PROGRAM MAIN
VAR
	bStartStop: BOOL := FALSE;
  bReset:     BOOL := FALSE;
  iCounter:   UINT := 0;
END_VAR

IF bStartStop THEN
  iCounter := iCounter+1;
END_IF

IF bReset THEN
  iCounter := 0;
END_IF

END_PROGRAM

(* stored: Version 1.1.0.1, ProductVersion 3.1.4024.0
   POU MAIN: Id {7ec64d65-0e79-432e-8ad8-0d9d00c3e123}, SpecialFunc None *)
